{attribute 'qualified_only'}
{attribute 'strict'}
TYPE ESvmRegressorType :
(
	EPS := TO_UDINT(ETcVnSvm.TCVN_SVM_EPS_REGRESSOR),
	NU := TO_UDINT(ETcVnSvm.TCVN_SVM_NU_REGRESSOR)
) UDINT;
END_TYPE

(* stored: Version 1.1.0.1, ProductVersion 3.1.4024.12
   DUT ESvmRegressorType: Id {b269595b-6bcc-49a1-9f45-7fbb49b3b97a} *)
